{attribute 'GeneratedUsingTerminal: ELX3351-0000-0016'}
{attribute addProperty BoxType "ELX3351-0000-0016"}
{attribute addProperty Description "ELX3351 1-channel precise load cell analysis, Ex i"}
{attribute addProperty Physics "KK"}
{attribute addProperty Id "RMB_StatusAT %I*RMB_Status_EE6B49B46RMB_Value_INT32AT %I*RMB_Value_INT_E9189C4B4RMB_ControlAT %Q*RMB_Control_4997AEF64WcStateAT %I*WcState_9091E0EB2InfoDataAT %I*InfoData_32EB74EA10"}
{attribute addProperty CRC "3746639915"}
{attribute addProperty Size "26"}
TYPE ELX3351_DF51302B EXTENDS EtcSlaveTerminalBase_947E5A46 :
STRUCT
	{attribute addProperty Name "RMB_Status"}
	RMB_Status : RMB_Status_EE6B49B4;
	{attribute addProperty Name "RMB_Value_INT32"}
	RMB_Value_INT32 : RMB_Value_INT_E9189C4B;
	{attribute addProperty Name "RMB_Control"}
	RMB_Control : RMB_Control_4997AEF6;
	{attribute addProperty Name "WcState"}
	WcState : WcState_9091E0EB;
	{attribute addProperty Name "InfoData"}
	InfoData : InfoData_32EB74EA;
END_STRUCT
END_TYPE

(* stored: Version 1.2.0.0, ProductVersion 3.1.4024.11
   DUT ELX3351_DF51302B: Id {d347f61b-6b81-4310-9d1e-0a9500509aa4} *)
